Staubli VAL3: readme.pgx

program readme()
begin
  //TITLE             : ATI force sensor
  //General desription: reads values from ATI force sensor with TCP/IP Socket interface
  //Hardware Required : ATI Force Sensor
  //Library Version   : 7.3.1
  //Public Variables  : bZero nForce nStatus
  //Public Program    : initialize() loopReadForce()
  //Included Libraries: None
  //Miscellaneous     : Requires a TCP/IP Client socket
  //Keywords          : ATI Force Sensor
end
